(* Logix 5000 project; controller VentiladorCamaraFriaParte1 vendor 1 type 14 code 89 rev 20.11; software revision 20.05 *)

TASK MainTask (continuous, watchdog 500 ms) : MainProgram

MODULES
   Controller : vendor 1 type 14 code 89 (CompactLogixL23E_QBFC1_Controller 0, rev 20.11)
      LocalENB : vendor 1 type 12 code 191 (CompactLogixL23E_QBFC1_Ethernet 1, rev 20.11)
      Local : CompactBus (CompactVirtualAdapter 3, rev 20.11)
         Discrete_Inputs : vendor 1 type 7 code 320 (Compact 1, rev 3.1, Input RPI 20 ms)
         Discrete_Outputs : vendor 1 type 7 code 322 (Compact 2, rev 3.1, Output RPI 20 ms)
         Analog_IO : vendor 1 type 10 code 120 (Compact 3, rev 1.1, Output RPI 80 ms)
         Counters : vendor 1 type 109 code 70 (Compact 4, rev 1.1, Output RPI 20 ms)
END_MODULES

PROGRAM MainProgram   (* main routine MainRoutine *)
VAR
   AcionaMotor : BOOL;
   AddTempoLig : ALIAS FOR Local:1:I.Data.6;
   BDMotor : BOOL;
   BSStartInversor : BOOL;
   Conta : COUNTER := (PRE := 10);
   ContaLigado : COUNTER;
   DecTempoLig : ALIAS FOR Local:1:I.Data.7;
   Desliga : ALIAS FOR Local:1:I.Data.0;
   Desligou : BOOL;
   Liga : ALIAS FOR Local:1:I.Data.1;
   MaquinaLigada : BOOL;
   Motor : ALIAS FOR Local:2:O.Data.1;
   SinalTempoMax : ALIAS FOR Local:2:O.Data.2;
   SinalTempoMin : ALIAS FOR Local:2:O.Data.3;
   SobrecargaInversor : ALIAS FOR Local:1:I.Data.2;
   StartInversor : BOOL;
   StopInversor : BOOL;
   TempoDesligado : TIMER := (PRE := 8000);
   TempoLigado : TIMER := (PRE := 5000);
   teste : COUNTER;
END_VAR

ROUTINE MainRoutine   (* ladder *)
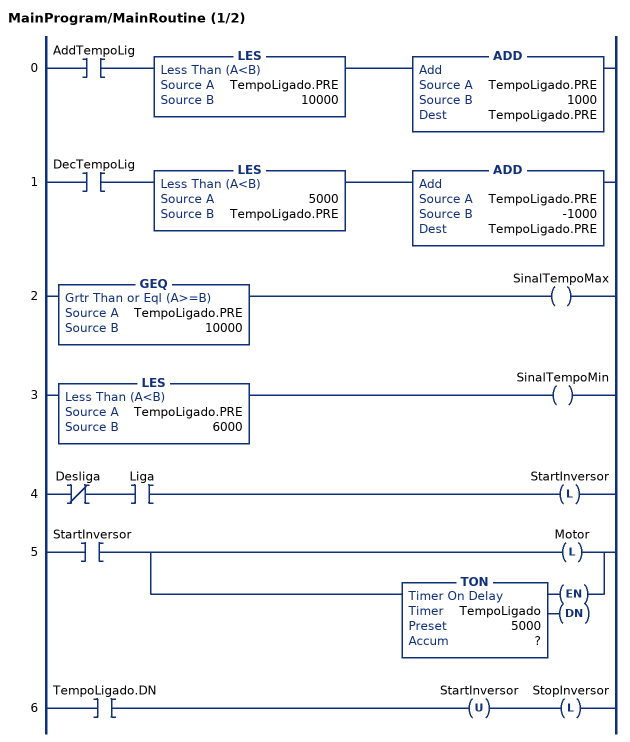
   0: XIC(AddTempoLig)LES(TempoLigado.PRE,10000)ADD(TempoLigado.PRE,1000,TempoLigado.PRE);
   1: XIC(DecTempoLig)LES(5000,TempoLigado.PRE)ADD(TempoLigado.PRE,-1000,TempoLigado.PRE);
   2: GEQ(TempoLigado.PRE,10000)OTE(SinalTempoMax);
   3: LES(TempoLigado.PRE,6000)OTE(SinalTempoMin);
   4: XIO(Desliga)XIC(Liga)OTL(StartInversor);
   5: XIC(StartInversor)[OTL(Motor) ,TON(TempoLigado,?,?) ];
   6: XIC(TempoLigado.DN)OTU(StartInversor)OTL(StopInversor);
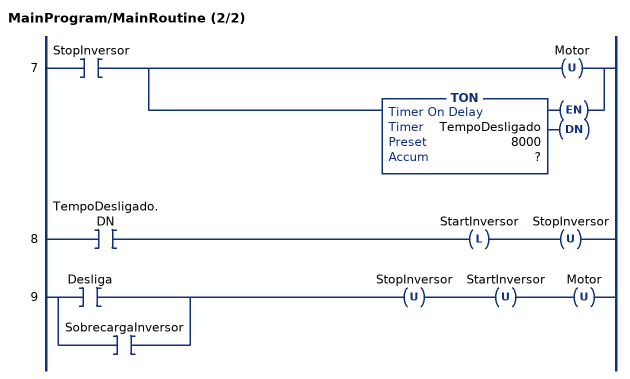
   7: XIC(StopInversor)[OTU(Motor) ,TON(TempoDesligado,?,?) ];
   8: XIC(TempoDesligado.DN)OTL(StartInversor)OTU(StopInversor);
   9: [XIC(Desliga) ,XIC(SobrecargaInversor) ]OTU(StopInversor)OTU(StartInversor)OTU(Motor);
END_ROUTINE
END_PROGRAM
